// TIA Portal V18 export
// export: Created 2026-03-12T15:56:20.3861378Z, ExportSetting WithDefaults, DisplayName Totally Integrated Automation Portal, DisplayVersion V18 Update 5, DisplayName TIA Portal Openness, DisplayVersion V18 Update 5, DisplayName TIA Portal Version Control Interface, DisplayVersion V18, DisplayName SINAMICS Startdrive Advanced, DisplayVersion V18, DisplayName SINAMICS Startdrive G130, G150, S120, S150, SINAMICS MV, S210, DisplayVersion V18, DisplayName SINAMICS Startdrive G110M, G120, G120C, G120D, G120P, G115D, DisplayVersion V18, DisplayName STEP 7 Professional, DisplayVersion V18 Update 5, DisplayName STEP 7 Safety, DisplayVersion V18, DisplayName WinCC Professional, DisplayVersion V18 Update 5
FUNCTION "PARTIDA_BOMBA_RESERVA_BH-01B" : Void   // FC66, LAD
{ S7_Optimized_Access := 'TRUE' }
VERSION : 0.1
// Network 1: Set memórias entradas digitais
// Network 2: Function Block FALHA
// Network 3: MODO AUTOMÁTICO: Condições para Modo Automático
// Network 4: Alternância/Rotatividade de bombas Principal-Reserva
// Network 5: Function Block CONDIÇÃO DE PARTIDA
// Network 6: Reset Comando Liga
// Network 7: Function Block MODOS DE OPERAÇÃO - Atribuição dos Modos de Operação
// Network 8: Intertravamento para habilitar o botão liga na IHM
// Network 9: Intertravamento de Segurança
// Network 10: Function Block SUCÇÃO OK
// Network 11: Aciona saída digital para partir o motor/bomba
// Network 12: Function Block HORÍMETRO - Tempo de bomba ligada em horas
// stored: AutoNumber true, IsIECCheckEnabled false, SetENOAutomatically false, UDAEnableTagReadback false
   VAR_TEMP   // added for the SCL form of the ladder/FBD networks
      _w1 : Bool;
   END_VAR
BEGIN

REGION Network 1: Set memórias entradas digitais
   // Instanciando entradas digitais em PLC Tags "M" Address
   // 
   // MODO LOCAL: Indica Operação Local da bomba
   // MODO LOCAL AUTO: Indicação de Funcionamento Local Automático
   // MODO REMOTO: Indica Operação Remoto da bomba (IHM)
   // LIGADO: Indica bomba ligada
   // FALHA: Sinal de Falha
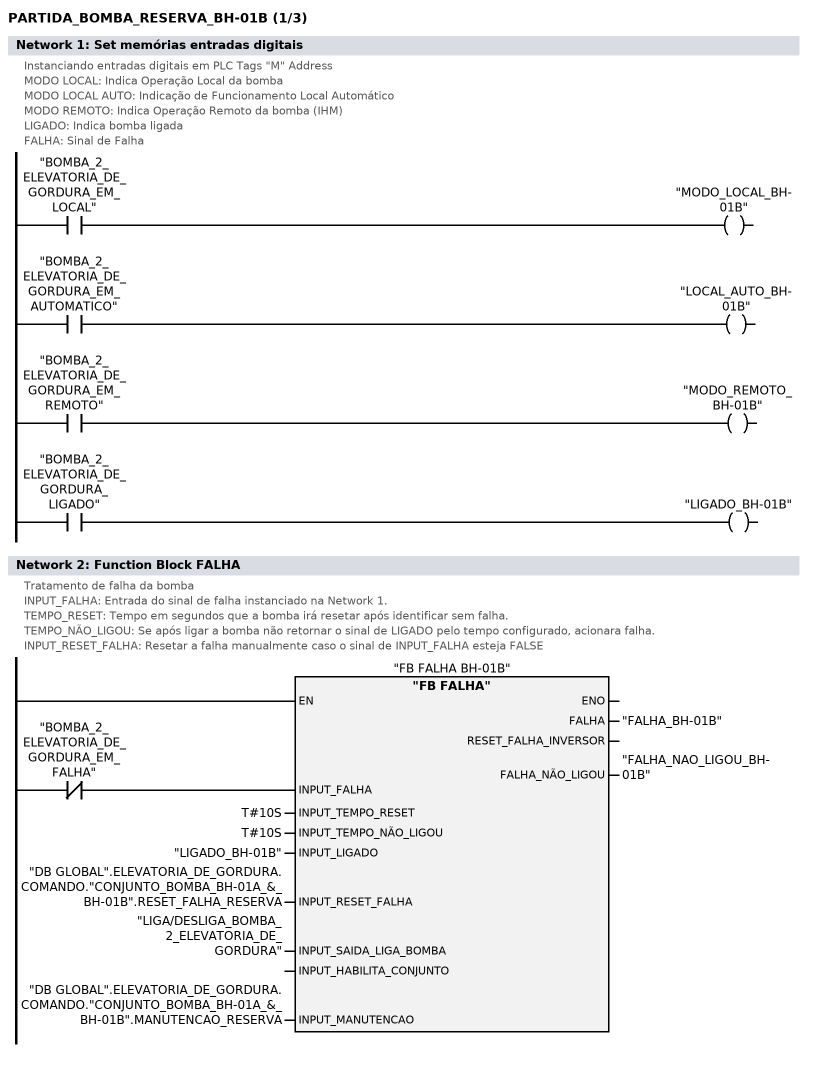
   RUNG wire#powerrail
      Contact( "BOMBA_2_ELEVATORIA_DE_GORDURA_EM_LOCAL" )
      Coil( "MODO_LOCAL_BH-01B" )
   END_RUNG
   RUNG wire#powerrail
      Contact( "BOMBA_2_ELEVATORIA_DE_GORDURA_EM_AUTOMATICO" )
      Coil( "LOCAL_AUTO_BH-01B" )
   END_RUNG
   RUNG wire#powerrail
      Contact( "BOMBA_2_ELEVATORIA_DE_GORDURA_EM_REMOTO" )
      Coil( "MODO_REMOTO_BH-01B" )
   END_RUNG
   RUNG wire#powerrail
      Contact( "BOMBA_2_ELEVATORIA_DE_GORDURA_LIGADO" )
      Coil( "LIGADO_BH-01B" )
   END_RUNG
   // the same network as SCL:
   "MODO_LOCAL_BH-01B" := "BOMBA_2_ELEVATORIA_DE_GORDURA_EM_LOCAL";
   "LOCAL_AUTO_BH-01B" := "BOMBA_2_ELEVATORIA_DE_GORDURA_EM_AUTOMATICO";
   "MODO_REMOTO_BH-01B" := "BOMBA_2_ELEVATORIA_DE_GORDURA_EM_REMOTO";
   "LIGADO_BH-01B" := "BOMBA_2_ELEVATORIA_DE_GORDURA_LIGADO";
END_REGION

REGION Network 2: Function Block FALHA
   // Tratamento de falha da bomba
   // INPUT_FALHA: Entrada do sinal de falha instanciado na Network 1.
   // TEMPO_RESET: Tempo em segundos que a bomba irá resetar após identificar sem falha.
   // TEMPO_NÃO_LIGOU: Se após ligar a bomba não retornar o sinal de LIGADO pelo tempo configurado, acionara falha.
   // INPUT_RESET_FALHA: Resetar a falha manualmente caso o sinal de INPUT_FALHA esteja FALSE
   RUNG wire#powerrail
      "FB FALHA BH-01B"(INPUT_FALHA := wire#w1, INPUT_TEMPO_RESET := T#10S, INPUT_TEMPO_NÃO_LIGOU := T#10S, INPUT_LIGADO := "LIGADO_BH-01B", INPUT_RESET_FALHA := "DB GLOBAL".ELEVATORIA_DE_GORDURA.COMANDO."CONJUNTO_BOMBA_BH-01A_&_BH-01B".RESET_FALHA_RESERVA, INPUT_SAIDA_LIGA_BOMBA := "LIGA/DESLIGA_BOMBA_2_ELEVATORIA_DE_GORDURA", INPUT_HABILITA_CONJUNTO :=, INPUT_MANUTENCAO := "DB GLOBAL".ELEVATORIA_DE_GORDURA.COMANDO."CONJUNTO_BOMBA_BH-01A_&_BH-01B".MANUTENCAO_RESERVA, FALHA => "FALHA_BH-01B", RESET_FALHA_INVERSOR =>, FALHA_NÃO_LIGOU => "FALHA_NAO_LIGOU_BH-01B")
   END_RUNG
   RUNG wire#powerrail
      I_Contact( "BOMBA_2_ ELEVATORIA_DE_GORDURA_EM_FALHA" )
   END_RUNG wire#w1
   // the same network as SCL:
   "FB FALHA BH-01B"(INPUT_FALHA := NOT "BOMBA_2_ ELEVATORIA_DE_GORDURA_EM_FALHA",   // "FB FALHA"
                     INPUT_TEMPO_RESET := T#10S,
                     INPUT_TEMPO_NÃO_LIGOU := T#10S,
                     INPUT_LIGADO := "LIGADO_BH-01B",
                     INPUT_RESET_FALHA := "DB GLOBAL".ELEVATORIA_DE_GORDURA.COMANDO."CONJUNTO_BOMBA_BH-01A_&_BH-01B".RESET_FALHA_RESERVA,
                     INPUT_SAIDA_LIGA_BOMBA := "LIGA/DESLIGA_BOMBA_2_ELEVATORIA_DE_GORDURA",
                     INPUT_MANUTENCAO := "DB GLOBAL".ELEVATORIA_DE_GORDURA.COMANDO."CONJUNTO_BOMBA_BH-01A_&_BH-01B".MANUTENCAO_RESERVA,
                     FALHA => "FALHA_BH-01B",
                     FALHA_NÃO_LIGOU => "FALHA_NAO_LIGOU_BH-01B");
END_REGION

REGION Network 3: MODO AUTOMÁTICO: Condições para Modo Automático
END_REGION

REGION Network 4: Alternância/Rotatividade de bombas Principal-Reserva
END_REGION

REGION Network 5: Function Block CONDIÇÃO DE PARTIDA
   // Varredura de condicionais para ligar
   // INPUT_LIGADO: Entrada do sinal de ligado instanciado na Network 1.
   // INPUT_FALHA: Entrada do sinal de falha da saída do bloco na Network 2.
   // INPUT_LOCAL: Entrada do sinal de modo local instanciado na Network 1.
   // INPUT_LOC_AUTO: Entrada do sinal do modo Local Automático
   // INPUT_REMOTO: Entrada do sinal de modo remoto instanciado na Network 1.
   // PARÂMETRO: Parâmetro de monitoramento para ligar e desligar a bomba em automático.
   // PARÂMETRO_LIGA/DESLIGA: Cadastros de programação liga/desliga em relação ao parâmetro.
   // CMD: Comandos recebidos pelo bloco
   // STATUS_MOTOR: Status de saída; 0 = DESLIGADO; 1 = LIGADO; 2 = FALHA; 3 = MANUTENÇÃO.
   // LIGA_BOMBA: Se TRUE, as condições estão OK para ligar na 5.
   // REMOTO_MAN: Saída indica que o motor/bomba está em modo Remoto Manual
   // REMOTO_AUTO: Saída indica que o motor/bomba está em modo Remoto Automático
   // LOCAL_MAN: Saída indica que o motor/bomba está em modo Local Manual
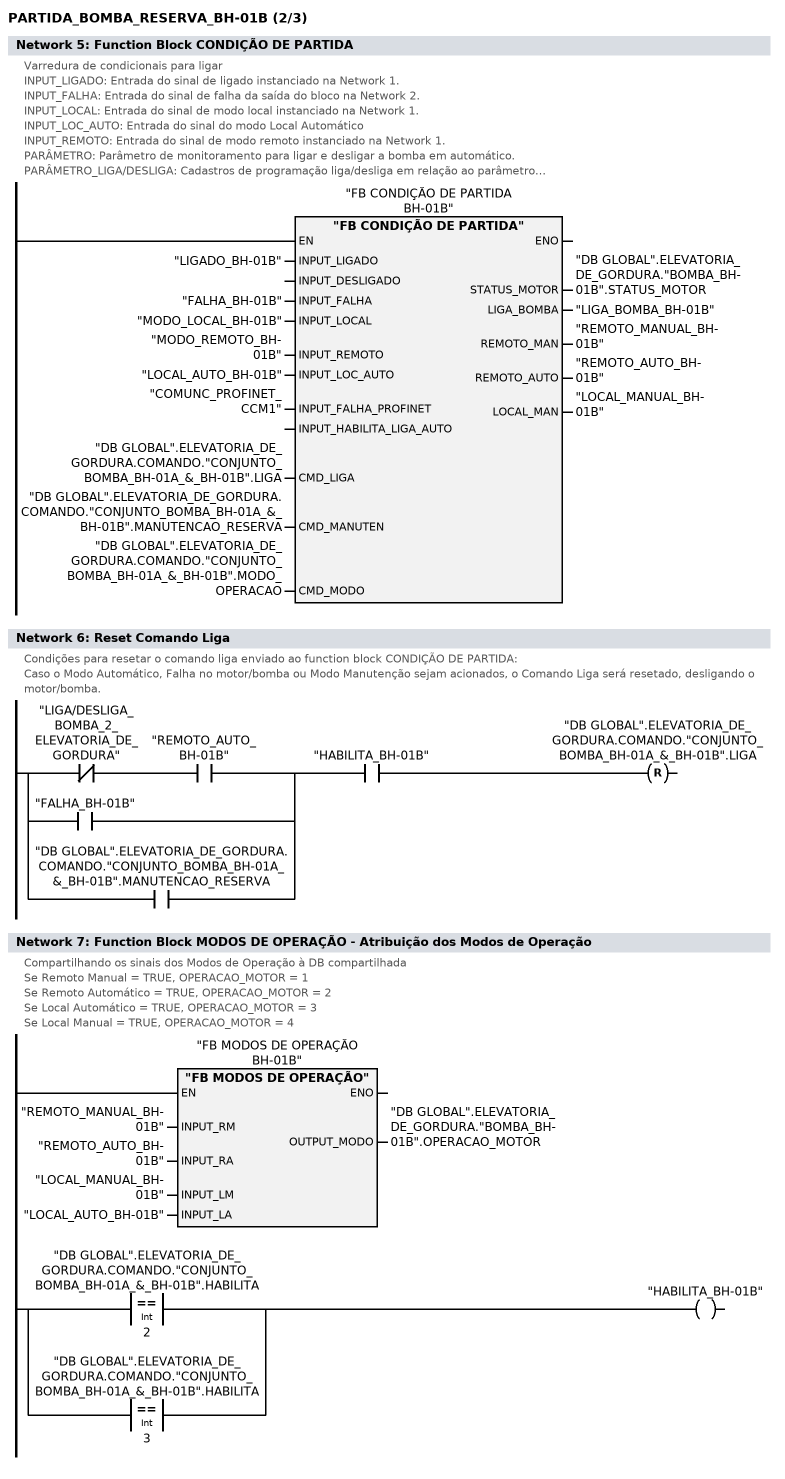
   RUNG wire#powerrail
      "FB CONDIÇÃO DE PARTIDA BH-01B"(INPUT_LIGADO := "LIGADO_BH-01B", INPUT_DESLIGADO :=, INPUT_FALHA := "FALHA_BH-01B", INPUT_LOCAL := "MODO_LOCAL_BH-01B", INPUT_REMOTO := "MODO_REMOTO_BH-01B", INPUT_LOC_AUTO := "LOCAL_AUTO_BH-01B", INPUT_FALHA_PROFINET := "COMUNC_PROFINET_CCM1", INPUT_HABILITA_LIGA_AUTO :=, CMD_LIGA := "DB GLOBAL".ELEVATORIA_DE_GORDURA.COMANDO."CONJUNTO_BOMBA_BH-01A_&_BH-01B".LIGA, CMD_MANUTEN := "DB GLOBAL".ELEVATORIA_DE_GORDURA.COMANDO."CONJUNTO_BOMBA_BH-01A_&_BH-01B".MANUTENCAO_RESERVA, CMD_MODO := "DB GLOBAL".ELEVATORIA_DE_GORDURA.COMANDO."CONJUNTO_BOMBA_BH-01A_&_BH-01B".MODO_OPERACAO, STATUS_MOTOR => "DB GLOBAL".ELEVATORIA_DE_GORDURA."BOMBA_BH-01B".STATUS_MOTOR, LIGA_BOMBA => "LIGA_BOMBA_BH-01B", REMOTO_MAN => "REMOTO_MANUAL_BH-01B", REMOTO_AUTO => "REMOTO_AUTO_BH-01B", LOCAL_MAN => "LOCAL_MANUAL_BH-01B")
   END_RUNG
   // the same network as SCL:
   "FB CONDIÇÃO DE PARTIDA BH-01B"(INPUT_LIGADO := "LIGADO_BH-01B",   // "FB CONDIÇÃO DE PARTIDA"
                           INPUT_FALHA := "FALHA_BH-01B",
                           INPUT_LOCAL := "MODO_LOCAL_BH-01B",
                           INPUT_REMOTO := "MODO_REMOTO_BH-01B",
                           INPUT_LOC_AUTO := "LOCAL_AUTO_BH-01B",
                           INPUT_FALHA_PROFINET := "COMUNC_PROFINET_CCM1",
                           CMD_LIGA := "DB GLOBAL".ELEVATORIA_DE_GORDURA.COMANDO."CONJUNTO_BOMBA_BH-01A_&_BH-01B".LIGA,
                           CMD_MANUTEN := "DB GLOBAL".ELEVATORIA_DE_GORDURA.COMANDO."CONJUNTO_BOMBA_BH-01A_&_BH-01B".MANUTENCAO_RESERVA,
                           CMD_MODO := "DB GLOBAL".ELEVATORIA_DE_GORDURA.COMANDO."CONJUNTO_BOMBA_BH-01A_&_BH-01B".MODO_OPERACAO,
                           STATUS_MOTOR => "DB GLOBAL".ELEVATORIA_DE_GORDURA."BOMBA_BH-01B".STATUS_MOTOR,
                           LIGA_BOMBA => "LIGA_BOMBA_BH-01B",
                           REMOTO_MAN => "REMOTO_MANUAL_BH-01B",
                           REMOTO_AUTO => "REMOTO_AUTO_BH-01B",
                           LOCAL_MAN => "LOCAL_MANUAL_BH-01B");
END_REGION

REGION Network 6: Reset Comando Liga
   // Condições para resetar o comando liga enviado ao function block CONDIÇÃO DE PARTIDA:
   // Caso o Modo Automático, Falha no motor/bomba ou Modo Manutenção sejam acionados, o Comando Liga será resetado, desligando o motor/bomba.
   RUNG wire#powerrail
      I_Contact( "LIGA/DESLIGA_BOMBA_2_ELEVATORIA_DE_GORDURA" )
      Contact( "REMOTO_AUTO_BH-01B" )
      wire#w1
      Contact( "HABILITA_BH-01B" )
      R_Coil( "DB GLOBAL".ELEVATORIA_DE_GORDURA.COMANDO."CONJUNTO_BOMBA_BH-01A_&_BH-01B".LIGA )
   END_RUNG
   RUNG wire#powerrail
      Contact( "FALHA_BH-01B" )
   END_RUNG wire#w1
   RUNG wire#powerrail
      Contact( "DB GLOBAL".ELEVATORIA_DE_GORDURA.COMANDO."CONJUNTO_BOMBA_BH-01A_&_BH-01B".MANUTENCAO_RESERVA )
   END_RUNG wire#w1
   // the same network as SCL:
   IF ((NOT "LIGA/DESLIGA_BOMBA_2_ELEVATORIA_DE_GORDURA" AND "REMOTO_AUTO_BH-01B") OR "FALHA_BH-01B" OR "DB GLOBAL".ELEVATORIA_DE_GORDURA.COMANDO."CONJUNTO_BOMBA_BH-01A_&_BH-01B".MANUTENCAO_RESERVA) AND "HABILITA_BH-01B" THEN
       "DB GLOBAL".ELEVATORIA_DE_GORDURA.COMANDO."CONJUNTO_BOMBA_BH-01A_&_BH-01B".LIGA := FALSE;
   END_IF;
END_REGION

REGION Network 7: Function Block MODOS DE OPERAÇÃO - Atribuição dos Modos de Operação
   // Compartilhando os sinais dos Modos de Operação à DB compartilhada
   // Se Remoto Manual = TRUE, OPERACAO_MOTOR = 1 
   // Se Remoto Automático = TRUE, OPERACAO_MOTOR = 2
   // Se Local Automático = TRUE, OPERACAO_MOTOR = 3
   // Se Local Manual = TRUE, OPERACAO_MOTOR = 4
   RUNG wire#powerrail
      "FB MODOS DE OPERAÇÃO BH-01B"(INPUT_RM := "REMOTO_MANUAL_BH-01B", INPUT_RA := "REMOTO_AUTO_BH-01B", INPUT_LM := "LOCAL_MANUAL_BH-01B", INPUT_LA := "LOCAL_AUTO_BH-01B", OUTPUT_MODO => "DB GLOBAL".ELEVATORIA_DE_GORDURA."BOMBA_BH-01B".OPERACAO_MOTOR)
   END_RUNG
   RUNG wire#powerrail
      { S7_Templates := "SrcType := Int" } EQ_Contact(in1 := "DB GLOBAL".ELEVATORIA_DE_GORDURA.COMANDO."CONJUNTO_BOMBA_BH-01A_&_BH-01B".HABILITA, in2 := 2)
      wire#w1
      Coil( "HABILITA_BH-01B" )
   END_RUNG
   RUNG wire#powerrail
      { S7_Templates := "SrcType := Int" } EQ_Contact(in1 := "DB GLOBAL".ELEVATORIA_DE_GORDURA.COMANDO."CONJUNTO_BOMBA_BH-01A_&_BH-01B".HABILITA, in2 := 3)
   END_RUNG wire#w1
   // the same network as SCL:
   "FB MODOS DE OPERAÇÃO BH-01B"(INPUT_RM := "REMOTO_MANUAL_BH-01B",   // "FB MODOS DE OPERAÇÃO"
                           INPUT_RA := "REMOTO_AUTO_BH-01B",
                           INPUT_LM := "LOCAL_MANUAL_BH-01B",
                           INPUT_LA := "LOCAL_AUTO_BH-01B",
                           OUTPUT_MODO => "DB GLOBAL".ELEVATORIA_DE_GORDURA."BOMBA_BH-01B".OPERACAO_MOTOR);
   "HABILITA_BH-01B" := ("DB GLOBAL".ELEVATORIA_DE_GORDURA.COMANDO."CONJUNTO_BOMBA_BH-01A_&_BH-01B".HABILITA = 2) OR ("DB GLOBAL".ELEVATORIA_DE_GORDURA.COMANDO."CONJUNTO_BOMBA_BH-01A_&_BH-01B".HABILITA = 3);
END_REGION

REGION Network 8: Intertravamento de Segurança
   // Caso a bomba esteja em REMOTO e a chave foi passada para LOCAL, A bomba é  colocada em modo REMOTO MANUAL E desligada. Desse modo, ao girar  novamente de LOCAL para REMOTO, é preciso que o  operador acione manualmente para ligar a bomba ou coloque manualmente em modo REMOTO AUTOMÁTICO. Isso acontece independente do estado em que a bomba se encontrava antes de girar de REMOTO para LOCAL, garantindo assim, segurança em casos de manutenção.
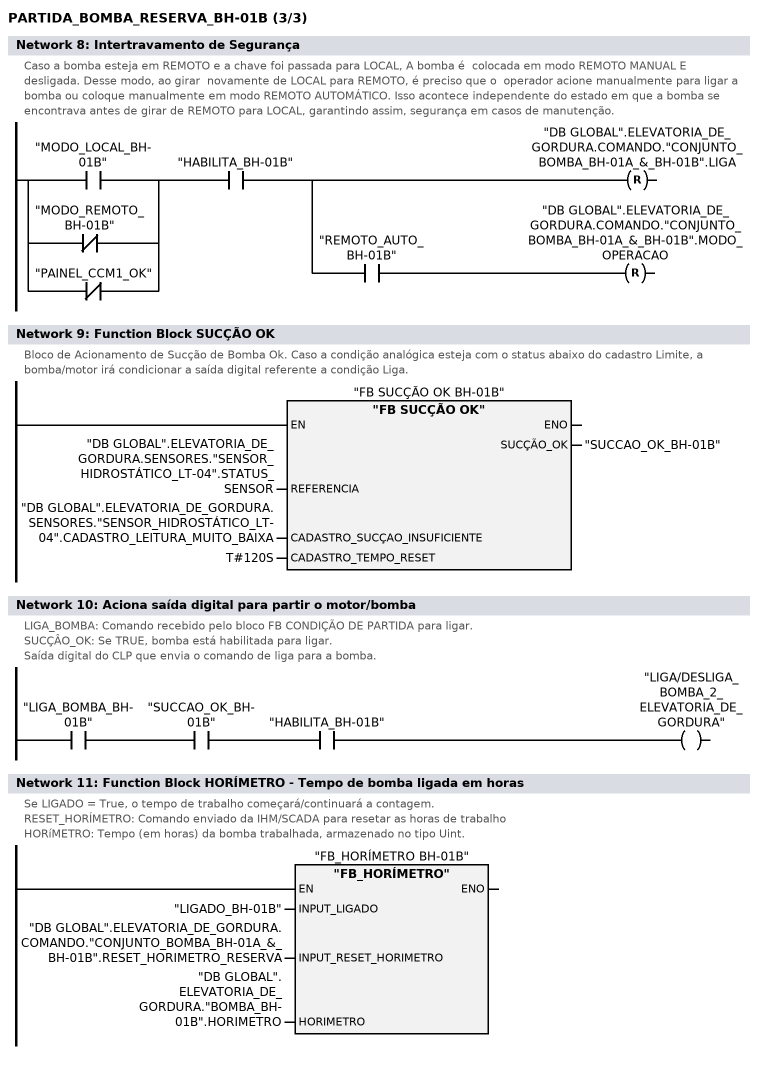
   RUNG wire#powerrail
      Contact( "MODO_LOCAL_BH-01B" )
      wire#w1
      Contact( "HABILITA_BH-01B" )
      wire#w2
      R_Coil( "DB GLOBAL".ELEVATORIA_DE_GORDURA.COMANDO."CONJUNTO_BOMBA_BH-01A_&_BH-01B".LIGA )
   END_RUNG
   RUNG wire#powerrail
      I_Contact( "MODO_REMOTO_BH-01B" )
   END_RUNG wire#w1
   RUNG wire#powerrail
      I_Contact( "PAINEL_CCM1_OK" )
   END_RUNG wire#w1
   RUNG wire#w2
      Contact( "REMOTO_AUTO_BH-01B" )
      R_Coil( "DB GLOBAL".ELEVATORIA_DE_GORDURA.COMANDO."CONJUNTO_BOMBA_BH-01A_&_BH-01B".MODO_OPERACAO )
   END_RUNG
   // the same network as SCL:
   #_w1 := ("MODO_LOCAL_BH-01B" OR NOT "MODO_REMOTO_BH-01B" OR NOT "PAINEL_CCM1_OK") AND "HABILITA_BH-01B";
   IF #_w1 THEN
       "DB GLOBAL".ELEVATORIA_DE_GORDURA.COMANDO."CONJUNTO_BOMBA_BH-01A_&_BH-01B".LIGA := FALSE;
   END_IF;
   IF #_w1 AND "REMOTO_AUTO_BH-01B" THEN
       "DB GLOBAL".ELEVATORIA_DE_GORDURA.COMANDO."CONJUNTO_BOMBA_BH-01A_&_BH-01B".MODO_OPERACAO := FALSE;
   END_IF;
END_REGION

REGION Network 9: Function Block SUCÇÃO OK
   // Bloco de Acionamento de Sucção de Bomba Ok. Caso a condição analógica esteja com o status abaixo do cadastro Limite, a bomba/motor irá condicionar a saída digital referente a condição Liga.
   RUNG wire#powerrail
      "FB SUCÇÃO OK BH-01B"(REFERENCIA := "DB GLOBAL".ELEVATORIA_DE_GORDURA.SENSORES."SENSOR_HIDROSTÁTICO_LT-04".STATUS_SENSOR, CADASTRO_SUCÇAO_INSUFICIENTE := "DB GLOBAL".ELEVATORIA_DE_GORDURA.SENSORES."SENSOR_HIDROSTÁTICO_LT-04".CADASTRO_LEITURA_MUITO_BAIXA, CADASTRO_TEMPO_RESET := T#120S, SUCÇÃO_OK => "SUCCAO_OK_BH-01B")
   END_RUNG
   // the same network as SCL:
   "FB SUCÇÃO OK BH-01B"(REFERENCIA := "DB GLOBAL".ELEVATORIA_DE_GORDURA.SENSORES."SENSOR_HIDROSTÁTICO_LT-04".STATUS_SENSOR,   // "FB SUCÇÃO OK"
                         CADASTRO_SUCÇAO_INSUFICIENTE := "DB GLOBAL".ELEVATORIA_DE_GORDURA.SENSORES."SENSOR_HIDROSTÁTICO_LT-04".CADASTRO_LEITURA_MUITO_BAIXA,
                         CADASTRO_TEMPO_RESET := T#120S,
                         SUCÇÃO_OK => "SUCCAO_OK_BH-01B");
END_REGION

REGION Network 10: Aciona saída digital para partir o motor/bomba
   // LIGA_BOMBA: Comando recebido pelo bloco FB CONDIÇÃO DE PARTIDA para ligar.
   // SUCÇÂO_OK: Se TRUE, bomba está habilitada para ligar.
   // 
   // Saída digital do CLP que envia o comando de liga para a bomba.
   RUNG wire#powerrail
      Contact( "LIGA_BOMBA_BH-01B" )
      Contact( "SUCCAO_OK_BH-01B" )
      Contact( "HABILITA_BH-01B" )
      Coil( "LIGA/DESLIGA_BOMBA_2_ELEVATORIA_DE_GORDURA" )
   END_RUNG
   // the same network as SCL:
   "LIGA/DESLIGA_BOMBA_2_ELEVATORIA_DE_GORDURA" := "LIGA_BOMBA_BH-01B" AND "SUCCAO_OK_BH-01B" AND "HABILITA_BH-01B";
END_REGION

REGION Network 11: Function Block HORÍMETRO - Tempo de bomba ligada em horas
   // Se LIGADO = True, o tempo de trabalho começará/continuará a contagem.
   // RESET_HORÍMETRO: Comando enviado da IHM/SCADA para resetar as horas de trabalho
   // HORíMETRO: Tempo (em horas) da bomba trabalhada, armazenado no tipo Uint.
   RUNG wire#powerrail
      "FB_HORÍMETRO BH-01B"(INPUT_LIGADO := "LIGADO_BH-01B", INPUT_RESET_HORIMETRO := "DB GLOBAL".ELEVATORIA_DE_GORDURA.COMANDO."CONJUNTO_BOMBA_BH-01A_&_BH-01B".RESET_HORIMETRO_RESERVA, HORIMETRO := "DB GLOBAL".ELEVATORIA_DE_GORDURA."BOMBA_BH-01B".HORIMETRO)
   END_RUNG
   // the same network as SCL:
   "FB_HORÍMETRO BH-01B"(INPUT_LIGADO := "LIGADO_BH-01B",   // "FB_HORÍMETRO"
                         INPUT_RESET_HORIMETRO := "DB GLOBAL".ELEVATORIA_DE_GORDURA.COMANDO."CONJUNTO_BOMBA_BH-01A_&_BH-01B".RESET_HORIMETRO_RESERVA,
                         HORIMETRO := "DB GLOBAL".ELEVATORIA_DE_GORDURA."BOMBA_BH-01B".HORIMETRO);
END_REGION
END_FUNCTION
